(* PLC project SafeLOGIC-1, BrAutomation SafeDESIGNER  4.3.2.11 *)
(* stored: companyURL http://www.br-automation.com, creationDateTime Mon Apr 16 08:26:33 2018 *)

PROGRAM Main

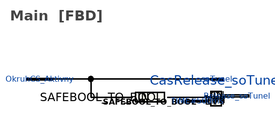
(* FBD diagram, written out as Structured Text *)
soTunel := OkruhCS_Aktivny;
CasRelease_soTunel(IN := SAFEBOOL_TO_BOOL(OkruhCS_Aktivny), PT := TIME#500ms);
Release_soTunel := CasRelease_soTunel.Q;
END_PROGRAM
